(* IEC 61131-3 sources: RAG_PLC/data/result/test/049, 2 files *)

(* ---- wrapped.st ---- *)
(* =========================================================
   Generated by PLC-Eval Benchmark Wrapper
   ========================================================= *)

FUNCTION_BLOCK LLM_Wrapper_FB
VAR_IN_OUT
    R_BUF : oscat_NETWORK_BUFFER;
    Xus_TN_SCREEN : us_TN_SCREEN;
END_VAR

VAR
    REQ_Size : UINT;
    REQ1 : BYTE;
    REQ2 : BYTE;
    REQ3 : BYTE;
END_VAR

Xus_TN_SCREEN.by_Input_ASCII_Code := BYTE#00;
Xus_TN_SCREEN.by_Input_Exten_Code := BYTE#00;

IF R_BUF.SIZE > UINT#0 THEN
    (* 解析接收到的数据 *)
    REQ_Size := R_BUF.SIZE;
    REQ1 := R_BUF.BUFFER[0];
    REQ2 := R_BUF.BUFFER[1];
    REQ3 := R_BUF.BUFFER[2];

    IF REQ1 = BYTE#27 AND REQ_Size >= UINT#3 THEN
        (* Escape *)
        IF REQ2 = BYTE#91 THEN
            (* 光标代码 *)
            IF (REQ3 >= BYTE#65 AND REQ3 <= BYTE#68) OR (REQ3 = BYTE#72) OR (REQ3 = BYTE#75) THEN
                Xus_TN_SCREEN.by_Input_Exten_Code := REQ3;
            END_IF;
        ELSIF REQ2 = BYTE#79 THEN
            IF REQ3 >= BYTE#80 AND REQ3 <= BYTE#83 THEN
                Xus_TN_SCREEN.by_Input_Exten_Code := REQ3;
            END_IF;
        END_IF;
    ELSIF REQ1 >= BYTE#32 AND REQ1 <= BYTE#126 THEN
        Xus_TN_SCREEN.by_Input_ASCII_Code := REQ1;
        Xus_TN_SCREEN.bo_Input_ASCII_IsNum := ISC_NUM(REQ1);
    ELSIF REQ1 = BYTE#8 OR REQ1 = BYTE#9 OR REQ1 = BYTE#13 OR REQ1 = BYTE#27 THEN
        Xus_TN_SCREEN.by_Input_Exten_Code := REQ1;
    END_IF;

    R_BUF.SIZE := UINT#00;
END_IF;
END_FUNCTION_BLOCK

PROGRAM Auto_Proxy_Prg
  VAR
    instance : LLM_Wrapper_FB;
  END_VAR

  instance();
END_PROGRAM

CONFIGURATION Config0
  RESOURCE Res0 ON PLC
    TASK TaskMain(INTERVAL := T#20ms, PRIORITY := 0);
    PROGRAM Inst0 WITH TaskMain : Auto_Proxy_Prg;
  END_RESOURCE
END_CONFIGURATION

(* ---- raw_code.st ---- *)
VAR_IN_OUT
    R_BUF : oscat_NETWORK_BUFFER;
    Xus_TN_SCREEN : us_TN_SCREEN;
END_VAR

VAR
    REQ_Size : UINT;
    REQ1 : BYTE;
    REQ2 : BYTE;
    REQ3 : BYTE;
END_VAR

Xus_TN_SCREEN.by_Input_ASCII_Code := BYTE#00;
Xus_TN_SCREEN.by_Input_Exten_Code := BYTE#00;

IF R_BUF.SIZE > UINT#0 THEN
    (* 解析接收到的数据 *)
    REQ_Size := R_BUF.SIZE;
    REQ1 := R_BUF.BUFFER[0];
    REQ2 := R_BUF.BUFFER[1];
    REQ3 := R_BUF.BUFFER[2];

    IF REQ1 = BYTE#27 AND REQ_Size >= UINT#3 THEN
        (* Escape *)
        IF REQ2 = BYTE#91 THEN
            (* 光标代码 *)
            IF (REQ3 >= BYTE#65 AND REQ3 <= BYTE#68) OR (REQ3 = BYTE#72) OR (REQ3 = BYTE#75) THEN
                Xus_TN_SCREEN.by_Input_Exten_Code := REQ3;
            END_IF;
        ELSIF REQ2 = BYTE#79 THEN
            IF REQ3 >= BYTE#80 AND REQ3 <= BYTE#83 THEN
                Xus_TN_SCREEN.by_Input_Exten_Code := REQ3;
            END_IF;
        END_IF;
    ELSIF REQ1 >= BYTE#32 AND REQ1 <= BYTE#126 THEN
        Xus_TN_SCREEN.by_Input_ASCII_Code := REQ1;
        Xus_TN_SCREEN.bo_Input_ASCII_IsNum := ISC_NUM(REQ1);
    ELSIF REQ1 = BYTE#8 OR REQ1 = BYTE#9 OR REQ1 = BYTE#13 OR REQ1 = BYTE#27 THEN
        Xus_TN_SCREEN.by_Input_Exten_Code := REQ1;
    END_IF;

    R_BUF.SIZE := UINT#00;
END_IF;
